PROGRAM PRG_Visualisierung
VAR_INPUT
	plot : ARRAY[1..GVL_Const.gc_max_Plots] OF REAL; 	//Array von den Werten (in REAL) die geplottet werden sollen
	TaskCycleTime_ms : UDINT;							//Zykluszeit in ms ( z.B. aus PRG_System)
END_VAR
VAR_OUTPUT
END_VAR
VAR
	
	fbpwmTrend :ARRAY[1..GVL_Const.gc_max_Plots] OF  FB_TrendBuffer;
	
	nindex:INT;
	
END_VAR


//Aufruf des FB zur Erzeugung des Trends
FOR nindex:=1  TO GVL_Const.gc_max_Plots DO  
	
	fbpwmTrend[nindex](
		uiValue:= plot[nindex],  						// Eingangssignal
		dtSystemTime:= PRG_System.GetSystemTime(), 
		tCycleTime:= UDINT_TO_TIME(TaskCycleTime_ms), 	// Zykluszeit
		bReverseFilll:= , 
		count=> , 
		dtFirstTimeStamp=> , 
		dtLastTimeStamp=> 
	);
END_FOR

END_PROGRAM

(* stored: Version 1.1.0.1, ProductVersion 3.1.4020.12
   POU PRG_Visualisierung: Id {27424455-d409-48d4-87e0-d9ff412f0a98}, SpecialFunc None *)
